{attribute 'OPC.UA.DA.StructuredType' := '1'}
TYPE ST_ElectricityMeterState :
STRUCT
	fPower			: REAL;
	sPowerUnit		: STRING := 'W';
	fWork			: REAL;
	sWorkUnit		: STRING := 'Wh';
END_STRUCT
END_TYPE

(* stored: Version 1.1.0.1, ProductVersion 3.1.4024.10
   DUT ST_ElectricityMeterState: Id {7d5a1323-3437-4d6e-9dc0-e12e1105ec4e} *)
